// TIA Portal V17 export
// export: Created 2024-09-02T12:50:15.7699467Z, ExportSetting WithDefaults, DisplayName Totally Integrated Automation Portal, DisplayVersion V17, DisplayName TIA Portal Openness, DisplayVersion V17, DisplayName TIA Portal Version Control Interface, DisplayVersion V17, DisplayName STEP 7 Professional, DisplayVersion V17, DisplayName STEP 7 Safety, DisplayVersion V17, DisplayName WinCC Professional, DisplayVersion V17
FUNCTION "AnwFC_ZP_SeriesError_OP70" : Void   // FC268, LAD
TITLE = Serial fault monitoring / Serienfehlerüberwachung
{ S7_Optimized_Access := 'TRUE' }
AUTHOR : OlegFuehrus
FAMILY : BA
NAME : BA
VERSION : 0.1
// stored: AutoNumber true, IsIECCheckEnabled false, SetENOAutomatically false, UDAEnableTagReadback false
   VAR_TEMP
      t_SerialFault_Start : Bool;
      t_SerialFault_available : Bool;
   END_VAR
   VAR CONSTANT
      Anzahl : Int := 3;
   END_VAR
   VAR_TEMP   // added for the SCL form of the ladder/FBD networks
      _w1 : Bool;
   END_VAR
BEGIN

REGION Network 1: Serie error active SLG1 / Serienfehlerauswertung aktiv
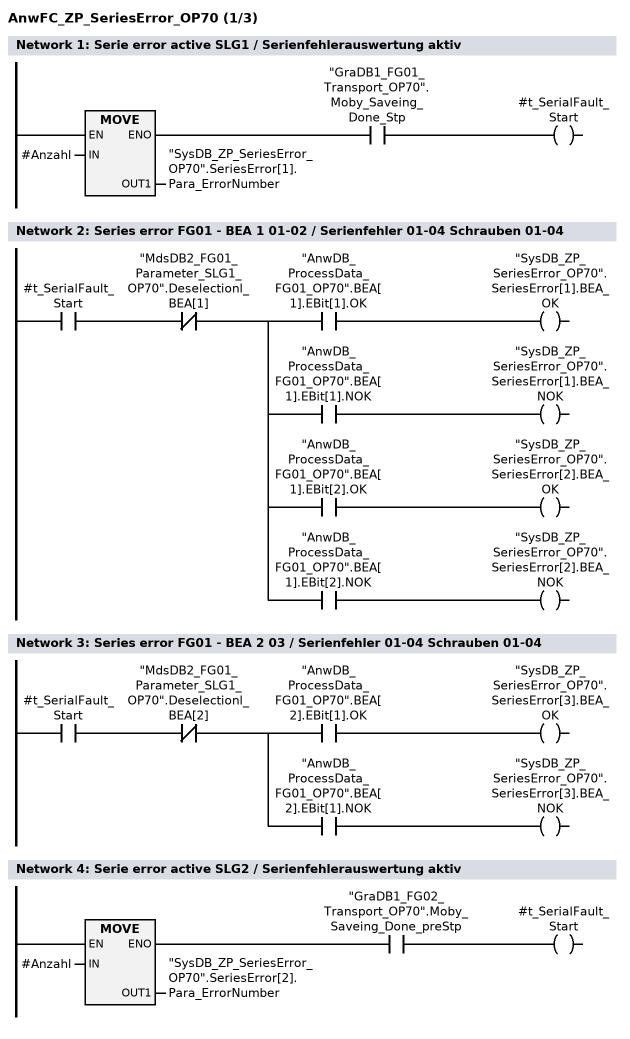
   RUNG wire#powerrail
      Move(in := #Anzahl, out1 => "SysDB_ZP_SeriesError_OP70".SeriesError[1].Para_ErrorNumber)
      Contact( "GraDB1_FG01_Transport_OP70".Moby_Saveing_Done_Stp )
      Coil( #t_SerialFault_Start )
   END_RUNG
   // the same network as SCL:
   "SysDB_ZP_SeriesError_OP70".SeriesError[1].Para_ErrorNumber := #Anzahl;
   #t_SerialFault_Start := "GraDB1_FG01_Transport_OP70".Moby_Saveing_Done_Stp;
END_REGION

REGION Network 2: Series error FG01 - BEA 1 01-02 / Serienfehler 01-04 Schrauben 01-04
   RUNG wire#powerrail
      Contact( #t_SerialFault_Start )
      I_Contact( "MdsDB2_FG01_Parameter_SLG1_OP70".Deselectionl_BEA[1] )
      wire#w1
      Contact( "AnwDB_ProcessData_FG01_OP70".BEA[1].EBit[1].OK )
      Coil( "SysDB_ZP_SeriesError_OP70".SeriesError[1].BEA_OK )
   END_RUNG
   RUNG wire#w1
      Contact( "AnwDB_ProcessData_FG01_OP70".BEA[1].EBit[1].NOK )
      Coil( "SysDB_ZP_SeriesError_OP70".SeriesError[1].BEA_NOK )
   END_RUNG
   RUNG wire#w1
      Contact( "AnwDB_ProcessData_FG01_OP70".BEA[1].EBit[2].OK )
      Coil( "SysDB_ZP_SeriesError_OP70".SeriesError[2].BEA_OK )
   END_RUNG
   RUNG wire#w1
      Contact( "AnwDB_ProcessData_FG01_OP70".BEA[1].EBit[2].NOK )
      Coil( "SysDB_ZP_SeriesError_OP70".SeriesError[2].BEA_NOK )
   END_RUNG
   // the same network as SCL:
   #_w1 := #t_SerialFault_Start AND NOT "MdsDB2_FG01_Parameter_SLG1_OP70".Deselectionl_BEA[1];
   "SysDB_ZP_SeriesError_OP70".SeriesError[1].BEA_OK := #_w1 AND "AnwDB_ProcessData_FG01_OP70".BEA[1].EBit[1].OK;
   "SysDB_ZP_SeriesError_OP70".SeriesError[1].BEA_NOK := #_w1 AND "AnwDB_ProcessData_FG01_OP70".BEA[1].EBit[1].NOK;
   "SysDB_ZP_SeriesError_OP70".SeriesError[2].BEA_OK := #_w1 AND "AnwDB_ProcessData_FG01_OP70".BEA[1].EBit[2].OK;
   "SysDB_ZP_SeriesError_OP70".SeriesError[2].BEA_NOK := #_w1 AND "AnwDB_ProcessData_FG01_OP70".BEA[1].EBit[2].NOK;
END_REGION

REGION Network 3: Series error FG01 - BEA 2 03 / Serienfehler 01-04 Schrauben 01-04
   RUNG wire#powerrail
      Contact( #t_SerialFault_Start )
      I_Contact( "MdsDB2_FG01_Parameter_SLG1_OP70".Deselectionl_BEA[2] )
      wire#w1
      Contact( "AnwDB_ProcessData_FG01_OP70".BEA[2].EBit[1].OK )
      Coil( "SysDB_ZP_SeriesError_OP70".SeriesError[3].BEA_OK )
   END_RUNG
   RUNG wire#w1
      Contact( "AnwDB_ProcessData_FG01_OP70".BEA[2].EBit[1].NOK )
      Coil( "SysDB_ZP_SeriesError_OP70".SeriesError[3].BEA_NOK )
   END_RUNG
   // the same network as SCL:
   #_w1 := #t_SerialFault_Start AND NOT "MdsDB2_FG01_Parameter_SLG1_OP70".Deselectionl_BEA[2];
   "SysDB_ZP_SeriesError_OP70".SeriesError[3].BEA_OK := #_w1 AND "AnwDB_ProcessData_FG01_OP70".BEA[2].EBit[1].OK;
   "SysDB_ZP_SeriesError_OP70".SeriesError[3].BEA_NOK := #_w1 AND "AnwDB_ProcessData_FG01_OP70".BEA[2].EBit[1].NOK;
END_REGION

REGION Network 4: Serie error active SLG2 / Serienfehlerauswertung aktiv
   RUNG wire#powerrail
      Move(in := #Anzahl, out1 => "SysDB_ZP_SeriesError_OP70".SeriesError[2].Para_ErrorNumber)
      Contact( "GraDB1_FG02_Transport_OP70".Moby_Saveing_Done_preStp )
      Coil( #t_SerialFault_Start )
   END_RUNG
   // the same network as SCL:
   "SysDB_ZP_SeriesError_OP70".SeriesError[2].Para_ErrorNumber := #Anzahl;
   #t_SerialFault_Start := "GraDB1_FG02_Transport_OP70".Moby_Saveing_Done_preStp;
END_REGION

REGION Network 5: Series error FG02 BEA 1 Ebit 04-09 / Serienfehler 01-04 Schrauben 01-04
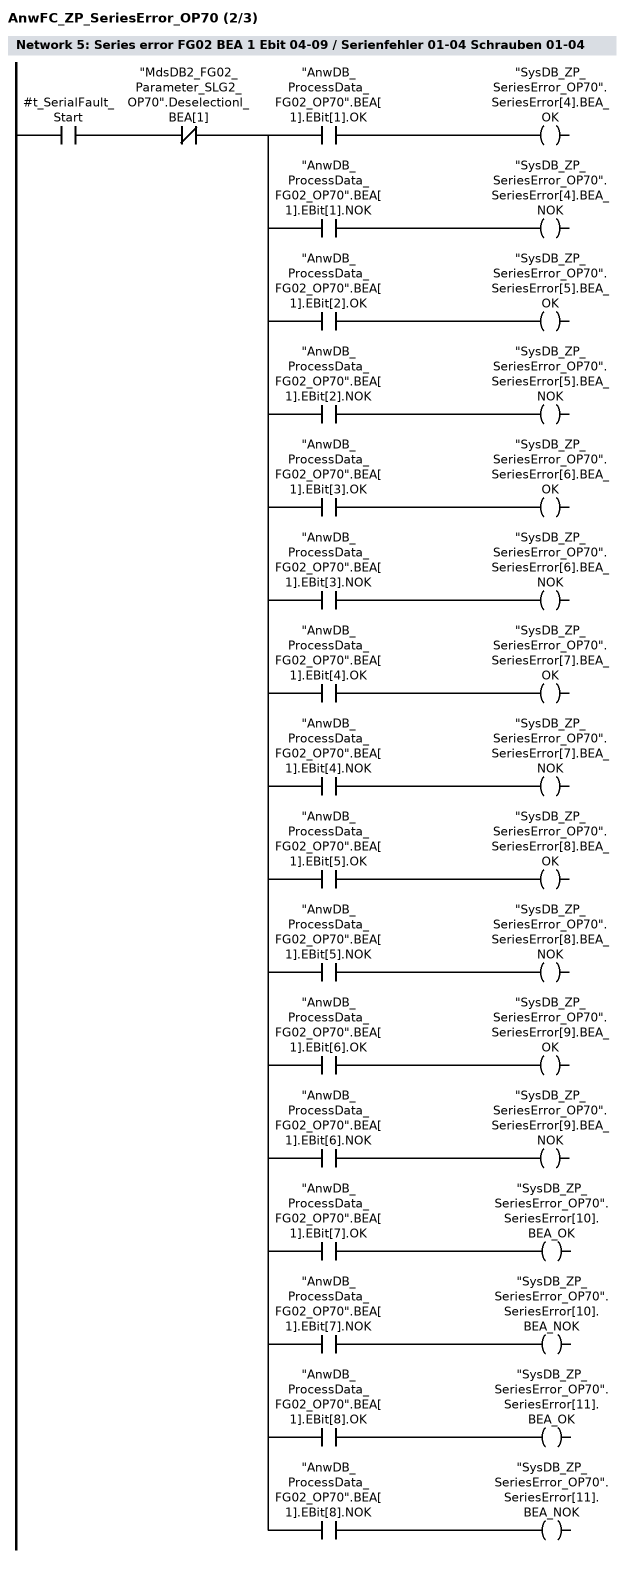
   RUNG wire#powerrail
      Contact( #t_SerialFault_Start )
      I_Contact( "MdsDB2_FG02_Parameter_SLG2_OP70".Deselectionl_BEA[1] )
      wire#w1
      Contact( "AnwDB_ProcessData_FG02_OP70".BEA[1].EBit[1].OK )
      Coil( "SysDB_ZP_SeriesError_OP70".SeriesError[4].BEA_OK )
   END_RUNG
   RUNG wire#w1
      Contact( "AnwDB_ProcessData_FG02_OP70".BEA[1].EBit[1].NOK )
      Coil( "SysDB_ZP_SeriesError_OP70".SeriesError[4].BEA_NOK )
   END_RUNG
   RUNG wire#w1
      Contact( "AnwDB_ProcessData_FG02_OP70".BEA[1].EBit[2].OK )
      Coil( "SysDB_ZP_SeriesError_OP70".SeriesError[5].BEA_OK )
   END_RUNG
   RUNG wire#w1
      Contact( "AnwDB_ProcessData_FG02_OP70".BEA[1].EBit[2].NOK )
      Coil( "SysDB_ZP_SeriesError_OP70".SeriesError[5].BEA_NOK )
   END_RUNG
   RUNG wire#w1
      Contact( "AnwDB_ProcessData_FG02_OP70".BEA[1].EBit[3].OK )
      Coil( "SysDB_ZP_SeriesError_OP70".SeriesError[6].BEA_OK )
   END_RUNG
   RUNG wire#w1
      Contact( "AnwDB_ProcessData_FG02_OP70".BEA[1].EBit[3].NOK )
      Coil( "SysDB_ZP_SeriesError_OP70".SeriesError[6].BEA_NOK )
   END_RUNG
   RUNG wire#w1
      Contact( "AnwDB_ProcessData_FG02_OP70".BEA[1].EBit[4].OK )
      Coil( "SysDB_ZP_SeriesError_OP70".SeriesError[7].BEA_OK )
   END_RUNG
   RUNG wire#w1
      Contact( "AnwDB_ProcessData_FG02_OP70".BEA[1].EBit[4].NOK )
      Coil( "SysDB_ZP_SeriesError_OP70".SeriesError[7].BEA_NOK )
   END_RUNG
   RUNG wire#w1
      Contact( "AnwDB_ProcessData_FG02_OP70".BEA[1].EBit[5].OK )
      Coil( "SysDB_ZP_SeriesError_OP70".SeriesError[8].BEA_OK )
   END_RUNG
   RUNG wire#w1
      Contact( "AnwDB_ProcessData_FG02_OP70".BEA[1].EBit[5].NOK )
      Coil( "SysDB_ZP_SeriesError_OP70".SeriesError[8].BEA_NOK )
   END_RUNG
   RUNG wire#w1
      Contact( "AnwDB_ProcessData_FG02_OP70".BEA[1].EBit[6].OK )
      Coil( "SysDB_ZP_SeriesError_OP70".SeriesError[9].BEA_OK )
   END_RUNG
   RUNG wire#w1
      Contact( "AnwDB_ProcessData_FG02_OP70".BEA[1].EBit[6].NOK )
      Coil( "SysDB_ZP_SeriesError_OP70".SeriesError[9].BEA_NOK )
   END_RUNG
   RUNG wire#w1
      Contact( "AnwDB_ProcessData_FG02_OP70".BEA[1].EBit[7].OK )
      Coil( "SysDB_ZP_SeriesError_OP70".SeriesError[10].BEA_OK )
   END_RUNG
   RUNG wire#w1
      Contact( "AnwDB_ProcessData_FG02_OP70".BEA[1].EBit[7].NOK )
      Coil( "SysDB_ZP_SeriesError_OP70".SeriesError[10].BEA_NOK )
   END_RUNG
   RUNG wire#w1
      Contact( "AnwDB_ProcessData_FG02_OP70".BEA[1].EBit[8].OK )
      Coil( "SysDB_ZP_SeriesError_OP70".SeriesError[11].BEA_OK )
   END_RUNG
   RUNG wire#w1
      Contact( "AnwDB_ProcessData_FG02_OP70".BEA[1].EBit[8].NOK )
      Coil( "SysDB_ZP_SeriesError_OP70".SeriesError[11].BEA_NOK )
   END_RUNG
   // the same network as SCL:
   #_w1 := #t_SerialFault_Start AND NOT "MdsDB2_FG02_Parameter_SLG2_OP70".Deselectionl_BEA[1];
   "SysDB_ZP_SeriesError_OP70".SeriesError[4].BEA_OK := #_w1 AND "AnwDB_ProcessData_FG02_OP70".BEA[1].EBit[1].OK;
   "SysDB_ZP_SeriesError_OP70".SeriesError[4].BEA_NOK := #_w1 AND "AnwDB_ProcessData_FG02_OP70".BEA[1].EBit[1].NOK;
   "SysDB_ZP_SeriesError_OP70".SeriesError[5].BEA_OK := #_w1 AND "AnwDB_ProcessData_FG02_OP70".BEA[1].EBit[2].OK;
   "SysDB_ZP_SeriesError_OP70".SeriesError[5].BEA_NOK := #_w1 AND "AnwDB_ProcessData_FG02_OP70".BEA[1].EBit[2].NOK;
   "SysDB_ZP_SeriesError_OP70".SeriesError[6].BEA_OK := #_w1 AND "AnwDB_ProcessData_FG02_OP70".BEA[1].EBit[3].OK;
   "SysDB_ZP_SeriesError_OP70".SeriesError[6].BEA_NOK := #_w1 AND "AnwDB_ProcessData_FG02_OP70".BEA[1].EBit[3].NOK;
   "SysDB_ZP_SeriesError_OP70".SeriesError[7].BEA_OK := #_w1 AND "AnwDB_ProcessData_FG02_OP70".BEA[1].EBit[4].OK;
   "SysDB_ZP_SeriesError_OP70".SeriesError[7].BEA_NOK := #_w1 AND "AnwDB_ProcessData_FG02_OP70".BEA[1].EBit[4].NOK;
   "SysDB_ZP_SeriesError_OP70".SeriesError[8].BEA_OK := #_w1 AND "AnwDB_ProcessData_FG02_OP70".BEA[1].EBit[5].OK;
   "SysDB_ZP_SeriesError_OP70".SeriesError[8].BEA_NOK := #_w1 AND "AnwDB_ProcessData_FG02_OP70".BEA[1].EBit[5].NOK;
   "SysDB_ZP_SeriesError_OP70".SeriesError[9].BEA_OK := #_w1 AND "AnwDB_ProcessData_FG02_OP70".BEA[1].EBit[6].OK;
   "SysDB_ZP_SeriesError_OP70".SeriesError[9].BEA_NOK := #_w1 AND "AnwDB_ProcessData_FG02_OP70".BEA[1].EBit[6].NOK;
   "SysDB_ZP_SeriesError_OP70".SeriesError[10].BEA_OK := #_w1 AND "AnwDB_ProcessData_FG02_OP70".BEA[1].EBit[7].OK;
   "SysDB_ZP_SeriesError_OP70".SeriesError[10].BEA_NOK := #_w1 AND "AnwDB_ProcessData_FG02_OP70".BEA[1].EBit[7].NOK;
   "SysDB_ZP_SeriesError_OP70".SeriesError[11].BEA_OK := #_w1 AND "AnwDB_ProcessData_FG02_OP70".BEA[1].EBit[8].OK;
   "SysDB_ZP_SeriesError_OP70".SeriesError[11].BEA_NOK := #_w1 AND "AnwDB_ProcessData_FG02_OP70".BEA[1].EBit[8].NOK;
END_REGION

REGION Network 6: Serie error active SLG3 / Serienfehlerauswertung aktiv
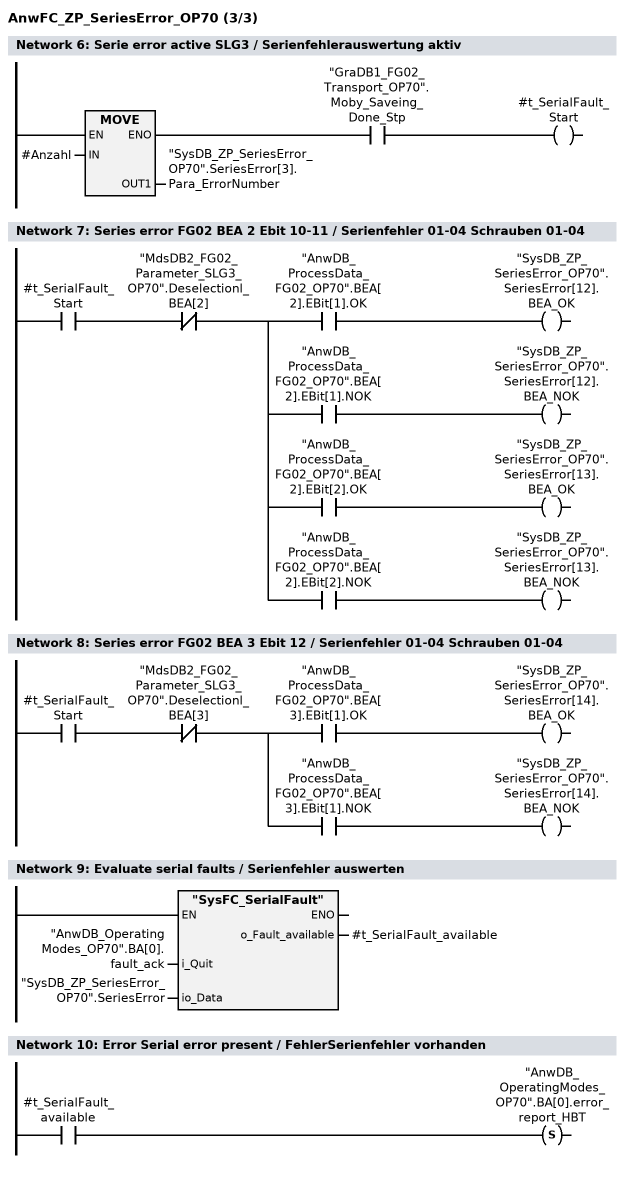
   RUNG wire#powerrail
      Move(in := #Anzahl, out1 => "SysDB_ZP_SeriesError_OP70".SeriesError[3].Para_ErrorNumber)
      Contact( "GraDB1_FG02_Transport_OP70".Moby_Saveing_Done_Stp )
      Coil( #t_SerialFault_Start )
   END_RUNG
   // the same network as SCL:
   "SysDB_ZP_SeriesError_OP70".SeriesError[3].Para_ErrorNumber := #Anzahl;
   #t_SerialFault_Start := "GraDB1_FG02_Transport_OP70".Moby_Saveing_Done_Stp;
END_REGION

REGION Network 7: Series error FG02 BEA 2 Ebit 10-11 / Serienfehler 01-04 Schrauben 01-04
   RUNG wire#powerrail
      Contact( #t_SerialFault_Start )
      I_Contact( "MdsDB2_FG02_Parameter_SLG3_OP70".Deselectionl_BEA[2] )
      wire#w1
      Contact( "AnwDB_ProcessData_FG02_OP70".BEA[2].EBit[1].OK )
      Coil( "SysDB_ZP_SeriesError_OP70".SeriesError[12].BEA_OK )
   END_RUNG
   RUNG wire#w1
      Contact( "AnwDB_ProcessData_FG02_OP70".BEA[2].EBit[1].NOK )
      Coil( "SysDB_ZP_SeriesError_OP70".SeriesError[12].BEA_NOK )
   END_RUNG
   RUNG wire#w1
      Contact( "AnwDB_ProcessData_FG02_OP70".BEA[2].EBit[2].OK )
      Coil( "SysDB_ZP_SeriesError_OP70".SeriesError[13].BEA_OK )
   END_RUNG
   RUNG wire#w1
      Contact( "AnwDB_ProcessData_FG02_OP70".BEA[2].EBit[2].NOK )
      Coil( "SysDB_ZP_SeriesError_OP70".SeriesError[13].BEA_NOK )
   END_RUNG
   // the same network as SCL:
   #_w1 := #t_SerialFault_Start AND NOT "MdsDB2_FG02_Parameter_SLG3_OP70".Deselectionl_BEA[2];
   "SysDB_ZP_SeriesError_OP70".SeriesError[12].BEA_OK := #_w1 AND "AnwDB_ProcessData_FG02_OP70".BEA[2].EBit[1].OK;
   "SysDB_ZP_SeriesError_OP70".SeriesError[12].BEA_NOK := #_w1 AND "AnwDB_ProcessData_FG02_OP70".BEA[2].EBit[1].NOK;
   "SysDB_ZP_SeriesError_OP70".SeriesError[13].BEA_OK := #_w1 AND "AnwDB_ProcessData_FG02_OP70".BEA[2].EBit[2].OK;
   "SysDB_ZP_SeriesError_OP70".SeriesError[13].BEA_NOK := #_w1 AND "AnwDB_ProcessData_FG02_OP70".BEA[2].EBit[2].NOK;
END_REGION

REGION Network 8: Series error FG02 BEA 3 Ebit 12 / Serienfehler 01-04 Schrauben 01-04
   RUNG wire#powerrail
      Contact( #t_SerialFault_Start )
      I_Contact( "MdsDB2_FG02_Parameter_SLG3_OP70".Deselectionl_BEA[3] )
      wire#w1
      Contact( "AnwDB_ProcessData_FG02_OP70".BEA[3].EBit[1].OK )
      Coil( "SysDB_ZP_SeriesError_OP70".SeriesError[14].BEA_OK )
   END_RUNG
   RUNG wire#w1
      Contact( "AnwDB_ProcessData_FG02_OP70".BEA[3].EBit[1].NOK )
      Coil( "SysDB_ZP_SeriesError_OP70".SeriesError[14].BEA_NOK )
   END_RUNG
   // the same network as SCL:
   #_w1 := #t_SerialFault_Start AND NOT "MdsDB2_FG02_Parameter_SLG3_OP70".Deselectionl_BEA[3];
   "SysDB_ZP_SeriesError_OP70".SeriesError[14].BEA_OK := #_w1 AND "AnwDB_ProcessData_FG02_OP70".BEA[3].EBit[1].OK;
   "SysDB_ZP_SeriesError_OP70".SeriesError[14].BEA_NOK := #_w1 AND "AnwDB_ProcessData_FG02_OP70".BEA[3].EBit[1].NOK;
END_REGION

REGION Network 9: Evaluate serial faults / Serienfehler auswerten
   RUNG wire#powerrail
      "SysFC_SerialFault"(i_Quit := "AnwDB_OperatingModes_OP70".BA[0].fault_ack, io_Data := "SysDB_ZP_SeriesError_OP70".SeriesError, o_Fault_available => #t_SerialFault_available)
   END_RUNG
   // the same network as SCL:
   "SysFC_SerialFault"(i_Quit := "AnwDB_OperatingModes_OP70".BA[0].fault_ack,
                       io_Data := "SysDB_ZP_SeriesError_OP70".SeriesError,
                       o_Fault_available => #t_SerialFault_available);
END_REGION

REGION Network 10: Error Serial error present / FehlerSerienfehler vorhanden
   RUNG wire#powerrail
      Contact( #t_SerialFault_available )
      S_Coil( "AnwDB_OperatingModes_OP70".BA[0].error_report_HBT )
   END_RUNG
   // the same network as SCL:
   IF #t_SerialFault_available THEN "AnwDB_OperatingModes_OP70".BA[0].error_report_HBT := TRUE; END_IF;
END_REGION
END_FUNCTION
